// TIA Portal V20 export
// export: Created 2025-12-01T14:56:07.6493265Z, ExportSetting None, DisplayName Totally Integrated Automation Portal, DisplayVersion V20 Update 3, DisplayName TIA Portal Openness, DisplayVersion V20 Update 3, DisplayName TIA Portal Version Control Interface, DisplayVersion V20 Update 3, DisplayName STEP 7 Professional, DisplayVersion V20 Update 3, DisplayName STEP 7 Safety, DisplayVersion V20 Update 2, DisplayName WinCC Basic/Comfort/Advanced, DisplayVersion V20 Update 3, DisplayName WinCC Professional, DisplayVersion V20 Update 3, DisplayName WinCC Unified, DisplayVersion V20 Update 3
TYPE "UDT_Informe_DatosUT"
   STRUCT
      MesaDestino : UInt;
      TipoCarga : UInt;
      Enfradado : UInt;
      Flejado : UInt;
      Etiquetado : UInt;
      CotaAltura : UInt;
      CotaAnchura : UInt;
      CotaLargura : UInt;
      Peso : UDInt;
      AtributosCarga : Struct
         Vacia : Bool;
         Pila : Bool;
         Remontada : Bool;
      END_STRUCT;
      PosEtiqueta : Struct
         Derecha : Bool;
         Izquierda : Bool;
      END_STRUCT;
      etiqueta : Array[0..42] of Char;
      EtiquetaRouter : UDInt;
   END_STRUCT;
END_TYPE
